// TwinCAT 3 PLC project Nepionic_Log
// Title: Nepionic_Log
// Company: Nepionic
// Author: Nepionic
// ProjectVersion: 0.1.1
// ProgramVersion: 3.1.4026.25
// libraries:
//   Tc2_Standard, * (Beckhoff Automation GmbH)
//   Tc2_System, * (Beckhoff Automation GmbH)
//   Tc2_Utilities, * (Beckhoff Automation GmbH)
//   Tc3_DynamicMemory, * (Beckhoff Automation GmbH)
// project tree:
//   Lib/Appenders/AdsLog/ AdsLogAppender.TcPOU, LogLevelToAdsLogMsgType.TcPOU (not stored)
//   Lib/Appenders/File/ DeleteFilesState.TcDUT (not stored), DeleteOldFiles.TcPOU (not stored), GenerateTimeData.TcPOU (not stored), GetFileAgeInSeconds.TcPOU (not stored), LoggingConfiguration.TcDUT (not stored), PersistToFileState.TcDUT (not stored), RollingIntervals.TcDUT
//   Lib/Appenders/ LogAppender.TcIO (not stored)
//   Lib/ Constants.TcGVL (not stored), DateTime.TcPOU (not stored), Error.TcDUT (not stored), ErrorCodes.TcDUT
//   Lib/Core/ LogAttribute.TcDUT (not stored), LogAttributeType.TcDUT (not stored), LogAttributeValueToString.TcPOU (not stored), LogLevel.TcDUT (not stored)
//   Lib/Manager/ GetLogManager.TcPOU (not stored), LogManager.TcPOU
//   Lib/Logger/ DefaultLogger.TcPOU (not stored), Logger.TcIO (not stored)
//   Lib/String/ AnyToString.TcPOU, DefaultStringBuilder.TcPOU (not stored), DynamicStringBuffer.TcPOU, LimitedStringBuilder.TcIO (not stored), StringBuilder.TcIO (not stored)

// ---- Lib/Appenders/File/RollingIntervals.TcDUT
/// Rolling interval to create a new log file when expired. 
{attribute 'qualified_only'}
{attribute 'strict'}
{attrivute 'to_string'}
TYPE RollingIntervals :
(
	None := 0,
	Hourly,
	Daily,
	Monthly
);
END_TYPE

// ---- Lib/ErrorCodes.TcDUT
/// Provides error codes for TcLogCore
{attribute 'qualified_only'}
{attribute 'strict'}
{attribute 'to_string'}
TYPE ErrorCodes : 
(
	None := 0,
	OpeningFileFailed,
	WritingToFileFailed,
	ClosingFileFailed,
	EnumeratingFilesInSpecifiedDirectoryFailed,
	DeletingFileFailed,
	FifoOverflow
);
END_TYPE

// ---- Lib/Appenders/AdsLog/AdsLogAppender.TcPOU
/// Log appender that writes to the TwinCAT ADS output window via `AdsLogStr`.
///
/// Register once at startup:
/// ```st
/// GetLogManager().Register(ads_appender);
/// ```
///
/// Optional: raise the threshold above DEBUG to reduce output noise:
/// ```st
/// ads_appender.Level := LogLevel.Warning;
/// ```
{attribute 'linkalways'}
{attribute 'no_explicit_call' := 'This FB is a CLASS and must be accessed using methods or properties'}
{attribute 'enable_dynamic_creation'}
FUNCTION_BLOCK PUBLIC AdsLogAppender IMPLEMENTS LogAppender
VAR
	_level : LogLevel := LogLevel.Debug;
END_VAR

METHOD Append : BOOL
VAR_INPUT
	level : LogLevel;
	message : Tc2_System.T_MaxString;
	source : Tc2_System.T_MaxString;
	attributes : ARRAY[0..9] OF LogAttribute;
	attribute_count : USINT;
END_VAR
VAR
	msg_type : DWORD;
	text : Tc2_System.T_MaxString;
	i : USINT;
	pair : Tc2_System.T_MaxString;
END_VAR
msg_type := Tc2_System.AdsLog_MsgType_Log OR LogLevelToAdsLogMsgType(level);

// Build: "[source] message  {key=value, ...}"
IF Tc2_Standard.Len(source) > 0 THEN
	text := Tc2_Standard.Concat('[', Tc2_Standard.Concat(source, '] '));
END_IF
text := Tc2_Standard.Concat(text, message);

IF attribute_count > 0 THEN
	text := Tc2_Standard.Concat(text, '  {');
	FOR i := 0 TO attribute_count - 1 DO
		IF i > 0 THEN
			text := Tc2_Standard.Concat(text, ', ');
		END_IF
		pair := Tc2_Standard.Concat(attributes[i].key, Tc2_Standard.Concat('=', LogAttributeValueToString(attributes[i])));
		text := Tc2_Standard.Concat(text, pair);
	END_FOR
	text := Tc2_Standard.Concat(text, '}');
END_IF

Tc2_System.AdsLogStr(msg_type, text, '');
Append := TRUE;
END_METHOD

{attribute 'monitoring' := 'call'}
PROPERTY Level : LogLevel
GET
Level := _level;
END_GET
SET
_level := Level;
END_SET
END_PROPERTY

END_FUNCTION_BLOCK

// ---- Lib/Manager/LogManager.TcPOU
/// Central log dispatcher.
/// Holds an ordered array of `LogAppender` sinks and fans out every record
/// to each appender whose `Level` threshold is satisfied.
///
/// Obtain the process-global singleton via `GetLogManager()` rather than
/// instantiating this directly.
///
/// Usage (startup — call once per appender before any log calls):
/// ```st
/// GetLogManager().Register(ads_appender);
/// GetLogManager().Register(otel_appender);
/// ```
{attribute 'linkalways'}
{attribute 'no_explicit_call' := 'This FB is a CLASS and must be accessed using methods or properties'}
{attribute 'enable_dynamic_creation'}
FUNCTION_BLOCK LogManager
VAR
	appenders : ARRAY[0..7] OF LogAppender;
	_count : UINT;
	dispatching : BOOL;
	_level : LogLevel := LogLevel.Debug;
END_VAR

/// Number of registered appenders (read-only, diagnostic).
{attribute 'monitoring' := 'call'}
PROPERTY PUBLIC Count : UINT
GET
Count := _count;
END_GET
END_PROPERTY

/// Fan a log record out to all registered appenders that meet the level threshold.
/// Guards against reentrancy (logging from inside an appender) and dispatches
/// nothing until at least one appender is registered.
METHOD PUBLIC Dispatch : BOOL
VAR_INPUT
	level : LogLevel;
	message : Tc2_System.T_MaxString;
	source : Tc2_System.T_MaxString;
	attributes : ARRAY[0..9] OF LogAttribute;
	attribute_count : USINT;
END_VAR
VAR
	i : UINT;
END_VAR
// Drop silently if no appenders registered yet (startup ordering safety)
IF _count = 0 THEN
	RETURN;
END_IF

// Reentrancy guard — an appender must never log back through the manager
IF dispatching THEN
	RETURN;
END_IF

// Global floor filter
IF level < _level THEN
	RETURN;
END_IF

dispatching := TRUE;

FOR i := 0 TO _count - 1 DO
	IF level >= appenders[i].Level THEN
		appenders[i].Append(level, message, source, attributes, attribute_count);
	END_IF
END_FOR

dispatching := FALSE;
Dispatch := TRUE;
END_METHOD

/// Global minimum level floor.
/// Records below this level are dropped before any per-appender check.
/// Defaults to `LogLevel.Debug` (pass everything to per-appender filters).
{attribute 'monitoring' := 'call'}
PROPERTY PUBLIC Level : LogLevel
GET // PUBLIC
Level := _level;
END_GET
SET // PUBLIC
_level := Level;
END_SET
END_PROPERTY

/// Register an appender with the log manager.
/// Up to 8 appenders are supported; extras are silently ignored.
/// Call once at startup before any log calls are made.
METHOD PUBLIC Register : BOOL
VAR_INPUT
	/// Appender instance to add (interface reference).
	appender : LogAppender;
END_VAR
IF _count >= 8 THEN
	RETURN;
END_IF

appenders[_count] := appender;
_count := _count + 1;
Register := TRUE;
END_METHOD

END_FUNCTION_BLOCK

// ---- Lib/String/AnyToString.TcPOU
/// Converts value of input data to string, where the input type can be any of 
/// the standard data types.
FUNCTION PUBLIC AnyToString : Tc2_System.T_MaxString
VAR_INPUT
	data : ANY;
END_VAR
VAR
	_any_byte : POINTER TO BYTE;
	_any_usint : POINTER TO USINT;
	_any_int : POINTER TO INT;
	_any_uint : POINTER TO UINT;
	_any_udInt : POINTER TO UDINT;
	_any_sint : POINTER TO SINT;
	_any_dint : POINTER TO DINT;
	_any_lint : POINTER TO LINT;
	_any_ulint : POINTER TO ULINT;
	_any_word : POINTER TO WORD;
	_any_lword : POINTER TO LWORD;
	_any_real : POINTER TO REAL;
	_any_lreal : POINTER TO LREAL;
	_any_date_and_time : POINTER TO DATE_AND_TIME;
	_any_date : POINTER TO DATE;
	_any_time : POINTER TO TIME;
	_any_wstring : POINTER TO WSTRING;
	_any_time_of_day : POINTER TO TOD;
	_any_string : POINTER TO STRING;
	_string : Tc2_System.T_MaxString;
	_wstring : WSTRING;
END_VAR

IF data.TypeClass = __SYSTEM.Type_Class.Type_Byte THEN
	_any_byte := data.pValue;
	AnyToString := BYTE_TO_STRING(_any_byte^);
ELSIF data.TypeClass = __SYSTEM.Type_Class.Type_Int THEN
	_any_int := data.pValue;
	AnyToString := INT_TO_STRING(_any_int^);
ELSIF data.TypeClass = __SYSTEM.Type_Class.Type_UInt THEN
	_any_uint := data.pValue;
	AnyToString := UINT_TO_STRING(_any_uint^);
ELSIF data.TypeClass = __SYSTEM.Type_Class.Type_UDint THEN
	_any_udint := data.pValue;
	AnyToString := UDINT_TO_STRING(_any_udint^);
ELSIF data.TypeClass = __SYSTEM.Type_Class.Type_SInt THEN
	_any_sint := data.pValue;
	AnyToString := SINT_TO_STRING(_any_sint^);
ELSIF data.TypeClass = __SYSTEM.Type_Class.Type_USint THEN
	_any_usint := data.pValue;
	AnyToString := USINT_TO_STRING(_any_usint^);
ELSIF data.TypeClass = __SYSTEM.Type_Class.Type_DInt THEN
	_any_dint := data.pValue;
	AnyToString := DINT_TO_STRING(_any_dint^);
ELSIF data.TypeClass = __SYSTEM.Type_Class.Type_LInt THEN
	_any_lint := data.pValue;
	AnyToString := LINT_TO_STRING(_any_lint^);
ELSIF data.TypeClass = __SYSTEM.Type_Class.Type_ULint THEN
	_any_ulint := data.pValue;
	AnyToString := ULINT_TO_STRING(_any_ulint^);
ELSIF data.TypeClass = __SYSTEM.Type_Class.Type_Word THEN
	_any_word := data.pValue;
	AnyToString := WORD_TO_STRING(_any_word^);
ELSIF data.TypeClass = __SYSTEM.Type_Class.Type_LWord THEN
	_any_lword := data.pValue;
	AnyToString := LWORD_TO_STRING(_any_lword^);
ELSIF data.TypeClass = __SYSTEM.Type_Class.Type_Real THEN
	_any_real := data.pValue;
	AnyToString := REAL_TO_STRING(_any_real^);
ELSIF data.TypeClass = __SYSTEM.Type_Class.Type_LReal THEN
	_any_lreal := data.pValue;
	AnyToString := LREAL_TO_STRING(_any_lreal^);
ELSIF data.TypeClass = __SYSTEM.Type_Class.Type_DateAndTime THEN
	_any_date_and_time := data.pValue;
	AnyToString := DT_TO_STRING(_any_date_and_time^);  
ELSIF data.TypeClass = __SYSTEM.Type_Class.Type_Date THEN
	_any_date := data.pValue;
	AnyToString := DATE_TO_STRING(_any_date^);
ELSIF data.TypeClass = __SYSTEM.Type_Class.Type_Time THEN
	_any_time := data.pValue;
	AnyToString := TIME_TO_STRING(_any_time^);
ELSIF data.TypeClass = __SYSTEM.Type_Class.Type_String THEN
	_any_string := data.pValue;
	AnyToString := _any_string^;
ELSIF data.TypeClass = __SYSTEM.Type_Class.Type_WString THEN
	_any_wstring := data.pValue;
	_wString := _any_wstring^;
	Tc2_Utilities.WSTRING_TO_STRING2(ADR(_string), ADR(_wstring), SIZEOF(_wstring));
	AnyToString := _string;
ELSIF data.TypeClass = __SYSTEM.Type_Class.Type_TimeOfDay THEN
	_any_time_of_day := data.pValue;
	AnyToString := TOD_TO_STRING(_any_time_of_day^);
ELSE
	AnyToString := TO_STRING(data.pValue^);
END_IF

END_FUNCTION

// ---- Lib/String/DynamicStringBuffer.TcPOU
{attribute 'hide_all_locals'}
FUNCTION_BLOCK INTERNAL DynamicStringBuffer
VAR_OUTPUT
	Error : Error; // Error information of this FB
END_VAR
VAR
	fifo : Tc2_Utilities.Fb_StringRingBuffer; // Necessary to buffer log data until it has been written to file.
	memory_manager : Tc3_DynamicMemory.Fb_DynMem_Manager; // Memory manager, required by DynMem_Buffer.
	dynamic_memory_buffer : Tc3_DynamicMemory.Fb_DynMem_Buffer(ipMemMan := memory_manager); // Provides dynamic buffer for Fifo. Is extended automatically if more than the
																   // default buffer size is needed.                  
	_busy : BOOL; // Buffer is busy; typically with writing data to the file system.
END_VAR

METHOD AddLine : BOOL
VAR_INPUT
	text : Tc2_System.T_MaxString; // Text to be added to the buffer
END_VAR
ResizeFifoBufferIfNecessary();
fifo.A_AddTail(putValue := Tc2_Standard.CONCAT(Tc2_Standard.LEFT(text, 254), '$N'));
END_METHOD

METHOD AddString : BOOL
VAR_INPUT
	text : Tc2_System.T_MaxString; // String to be added to the buffer
END_VAR
ResizeFifoBufferIfNecessary();
fifo.A_AddTail(putValue := text);
END_METHOD

METHOD PRIVATE AllocateBuffer : BOOL // Allocates buffer FOR the fifo.
VAR_INPUT
	bufferSize : UDINT; // Initial buffer size in BYTEs for fifo buffer.
END_VAR
dynamic_memory_buffer.CreateBuffer(nSize:=bufferSize, bReset:=TRUE);
fifo.pBuffer := dynamic_memory_buffer.pBuffer;
fifo.cbBuffer := bufferSize;
END_METHOD

{attribute 'monitoring':='call'}
PROPERTY PUBLIC Busy : BOOL
GET // PUBLIC
Busy := _busy;
END_GET
SET // PRIVATE
_busy := Busy;
END_SET
END_PROPERTY

METHOD FB_exit : BOOL
VAR_INPUT
	bInCopyCode : BOOL; // if TRUE, the exit method is called for exiting an instance that is copied afterwards (online change).
END_VAR
dynamic_memory_buffer.Clear();
END_METHOD

METHOD FlushCache : BOOL
fifo.A_Reset();
END_METHOD

METHOD INTERNAL Init : BOOL
VAR_INPUT
	bufferSize : UDINT; // Initial buffer size in BYTEs for fifo buffer.
END_VAR
AllocateBuffer(bufferSize);
END_METHOD

{attribute 'hide_all_locals'}
METHOD PersistToFile : BOOL
VAR_INPUT
	enable: BOOL; // TRUE starts persistence mechanism
	fileName : Tc2_System.T_MaxString; // File name including its path
END_VAR
VAR_INST
	state : PersistToFileState;
	
	file_open : Tc2_System.FB_FileOpen;
	file_handle : UINT;
	
	file_write : Tc2_System.FB_FileWrite;
	lockFileWriteToForceRisingEdge : BOOL; // filePuts can only be executed every other cycle
										 // since it needs a rising edge to execute.
	file_close : Tc2_System.FB_FileClose;
	
	buffer : ARRAY[0..Constants.BufferSize] OF BYTE;
	currentBufferPos : UDINT;
	fifo_head_string : Tc2_System.T_MaxString;
	fifo_head_length : UDINT;
	fifo_head_bytes : ARRAY[0..Tc2_System.Max_String_Length] OF BYTE;
	i : UINT;
END_VAR
VAR CONSTANT
	NetId : STRING := '';
	Timeout : TIME := Tc2_System.Default_Ads_Timeout;
	MaxLogsPerCycle : UINT := UDINT_TO_UINT(Constants.BufferSize / Tc2_System.Max_String_Length);
	MaxBufferPosition : UDINT := SIZEOF(buffer) - Tc2_System.Max_String_Length;
END_VAR
// State machine
// Using if-statements instead of case for performance reasons:
// Some states execute instantly and allow thus the next state 
// to start within the same plc cycle.

// *** I D L E ***
IF state = PersistToFileState.Idle THEN
	lockFileWriteToForceRisingEdge := FALSE;
	IF fifo.nCount > 0 AND enable THEN 
		lockFileWriteToForceRisingEdge := FALSE;
		state := PersistToFileState.OpenFile;
	END_IF
END_IF
    
// *** O P E N   F I L E ***
file_open(
	sNetId := NetId,
	sPathName := fileName,
	nMode := Tc2_System.Fopen_ModeAppend OR Tc2_System.Fopen_ModeText, 
	ePath := Tc2_System.Path_Generic,
	bExecute := (state = PersistToFileState.OpenFile),
	tTimeout := Timeout,
	hFile => file_handle
);

IF state = PersistToFileState.OpenFile THEN
	IF file_open.bError THEN
		state := PersistToFileState.CloseFile;
	ELSIF NOT file_open.bBusy THEN
		state := PersistToFileState.GetStringFromFifo; 
	END_IF
END_IF 

// *** P O P   F R O M   F I F O ***
IF state = PersistToFileState.GetStringFromFifo THEN
	IF NOT lockFileWriteToForceRisingEdge THEN
		currentBufferPos := 0;
		FOR i:=0 TO MaxLogsPerCycle DO
			IF fifo.nCount <= 0 THEN EXIT; END_IF
			IF currentBufferPos >= MaxBufferPosition THEN EXIT; END_IF
			
			fifo.A_RemoveHead(getValue => fifo_head_string); 
			fifo_head_bytes := Tc2_Utilities.MaxString_To_ByteArr(fifo_head_string);
			fifo_head_length := INT_TO_UDINT(Tc2_System.Len(fifo_head_string));
			Tc2_System.MemCpy(
				destAddr := ADR(buffer) + SIZEOF(BYTE) * currentBufferPos,
				srcAddr := ADR(fifo_head_bytes),
				n := fifo_head_length
			);    
			currentBufferPos := currentBufferPos + fifo_head_length;  
		END_FOR
		state := PersistToFileState.AppendDataToFile;
	END_IF
	lockFileWriteToForceRisingEdge := FALSE;
END_IF
  
// *** W R I T E   T O   F I L E ***
file_write(
	sNetId := NetId, 
	hFile := file_handle, 
	pWriteBuff := ADR(buffer),
	cbWriteLen := currentBufferPos,
	bExecute := state = PersistToFileState.AppendDataToFile, 
	tTimeout := Timeout
); 

IF state = PersistToFileState.AppendDataToFile THEN
	lockFileWriteToForceRisingEdge := TRUE;   
	IF file_write.bError THEN
		state := PersistToFileState.CloseFile;
	ELSIF fifo.nCount > 0 AND NOT file_write.bBusy THEN
		state := PersistToFileState.GetStringFromFifo; 
	ELSIF fifo.nCount = 0 THEN
		state := PersistToFileState.CloseFile;
	END_IF
END_IF
    
// *** C L O S E   F I L E ***
file_close(
	sNetId := NetId,
	hFile := file_handle, 
	bExecute := (state = PersistToFileState.CloseFile),
	tTimeout := Timeout
);

IF state = PersistToFileState.CloseFile THEN
	IF NOT file_close.bBusy THEN
		state := PersistToFileState.Idle;
	END_IF
END_IF

// Close file in case of error
IF file_open.bError THEN
	state := PersistToFileState.CloseFile;
END_IF

IF file_write.bError THEN
	state := PersistToFileState.CloseFile;
END_IF

IF NOT fifo.bOk
	AND fifo.nCount > 0
	AND state <> PersistToFileState.Idle
THEN 
  state := PersistToFileState.CloseFile; 
END_IF

// Error handling
IF file_open.bError THEN
  Error.Active := TRUE;
  Error.Code := ErrorCodes.OpeningFileFailed;
  Error.Info := Tc2_Standard.ConCat('Opening file failed. Error thrown by FB_FileOpen. Consult Beckhoff InfoSys. Internal Error: ', UDINT_TO_STRING(file_open.nErrId));
ELSIF file_write.bError THEN
  Error.Active := TRUE;
  Error.Code := ErrorCodes.WritingToFileFailed;
  Error.Info := Tc2_Standard.ConCat('Writing to file failed. Error thrown by FB_FileWrite. Consult Beckhoff InfoSys. Internal Error: ', UDINT_TO_STRING(file_write.nErrId));
ELSIF file_close.bError THEN
  Error.Active := TRUE;
  Error.Code := ErrorCodes.ClosingFileFailed;
  Error.Info := Tc2_Standard.ConCat('Closing file failed. Error thrown by FB_FileClose. Consult Beckhoff InfoSys. Internal Error: ', UDINT_TO_STRING(file_close.nErrId));
ELSIF NOT fifo.bOk AND fifo.nCount > 0 THEN
  Error.Active := TRUE;
  Error.Code := ErrorCodes.FifoOverflow;
  Error.Info := 'FIFO overflow. Check if plc has enough free memory.';
ELSE
  Error.Active := FALSE;
  Error.Code := ErrorCodes.None;
  Error.Info := '';
END_IF

// Set busy state
Busy := (state <> PersistToFileState.Idle OR fifo.nCount > 0);

(* Uncomment for cyclic logging of state machine, buffer usage & errors

ADSLOGSTR(ADSLOG_MSGTYPE_LOG, 
  Tc2_Standard.CONCAT('****DynamicStringBuffer.state:', 
  Tc2_Standard.CONCAT(UINT_TO_STRING(state),
  Tc2_Standard.CONCAT(', DynamicStringBuffer.hFile:', UINT_TO_STRING(hFile)))), '');

ADSLOGSTR(ADSLOG_MSGTYPE_LOG, 
  Tc2_Standard.CONCAT('****Fifo: used ', 
  Tc2_Standard.CONCAT(UDINT_TO_STRING(Fifo.cbSize),
  Tc2_Standard.CONCAT(' of ', UDINT_TO_STRING(Fifo.cbBuffer)))), '');
  
IF Error.Active THEN
  ADSLOGSTR(ADSLOG_MSGTYPE_LOG, 
    Tc2_Standard.CONCAT('****DynamicStringBuffer.Error: ', Error.Info), 
    '');  
END_IF
*)
END_METHOD

METHOD PopHead : Tc2_System.T_MaxString
VAR_INST
	headString : Tc2_System.T_MaxString;
END_VAR
fifo.A_RemoveHead(getValue => headString);
PopHead := headString;
END_METHOD

// Resizes the buffer for the FIFO if necessary
METHOD PRIVATE ResizeFifoBufferIfNecessary : BOOL
VAR
	requiredSize : UDINT;
	newSize : DINT;
END_VAR
requiredSize := fifo.cbSize + (Tc2_System.MAX_STRING_LENGTH + Constants.FifoOverhead);

IF requiredSize > fifo.cbBuffer THEN
	dynamic_memory_buffer.Resize(nSize := requiredSize*SIZEOF(BYTE), bPreserve:=TRUE, bReset:=TRUE);
	fifo.pBuffer := dynamic_memory_buffer.pBuffer;
	fifo.cbBuffer := requiredSize;
END_IF
END_METHOD

END_FUNCTION_BLOCK
